{attribute 'GeneratedUsingTerminal: EL7342-0000-0016'}
{attribute addProperty BoxType "EL7342-0000-0016"}
{attribute addProperty Id "ControlAT %Q*Control_F189B7373Set_counter_valueAT %Q*UINT2"}
{attribute addProperty CRC "780319811"}
{attribute addProperty Size "5"}
TYPE ENC_Control_compact_Channel_2E82BC43 EXTENDS OutputBase_10CEE7DE :
STRUCT
	{attribute addProperty Name "Control"}
	Control AT %Q* : Control_F189B737;
	{attribute addProperty Name "Set_counter_value"}
	Set_counter_value AT %Q* : UINT;
END_STRUCT
END_TYPE

(* stored: Version 1.2.0.0, ProductVersion 3.1.4024.11
   DUT ENC_Control_compact_Channel_2E82BC43: Id {c509c475-3de3-47d0-9a24-6144a467a31d} *)
